PROGRAM MAIN
VAR
	T1: TON;
END_VAR

T1(IN:=GVL1.Switch , PT:=T#5s , Q=>GVL1.Lamp );

END_PROGRAM

(* stored: Version 1.1.0.1, ProductVersion 3.1.4024.5
   POU MAIN: Id {0ac9e51b-c44e-44a0-8454-c4e92c9a0fca}, SpecialFunc None *)
